TYPE CmpCore :
STRUCT
	
	Framework: Framework;

END_STRUCT
END_TYPE

(* stored: Version 1.1.0.1, ProductVersion 3.1.4024.6
   DUT CmpCore: Id {b5439e86-14d1-454e-a435-6a7432a30d74} *)
